// TIA Portal V17 export
// export: Created 2022-07-05T08:45:17.4289241Z, ExportSetting WithDefaults, DisplayName Totally Integrated Automation Portal, DisplayVersion V17, DisplayName TIA Portal Openness, DisplayVersion V17, DisplayName TIA Portal Version Control Interface, DisplayVersion V17, DisplayName STEP 7 Professional, DisplayVersion V17, DisplayName STEP 7 Safety, DisplayVersion V17, DisplayName WinCC Advanced, DisplayVersion V17
TYPE "typeFbDiagnostics"
TITLE = typeDiagnosticsFBTemplate
// stored: IsFailsafeCompliant false
   STRUCT
      status : Word;   // Status of the FB or error identification when error occurred
      subfunctionStatus : DWord;   // Status or return value of called FBs, FCs and system blocks
   END_STRUCT;
END_TYPE
